PROGRAM Systemzeit
VAR
	fbFB_LocalSystemTime: FB_LocalSystemTime;
	fbGETSYSTEMTIME		: GETSYSTEMTIME;
    sNetID     			: T_AmsNetID := '';
    bEnable    			: BOOL := 1;
    dwCycle    			: DWORD(1..86400) := 5;
    dwOpt      			: DWORD := 1;
    tTimeout   			: TIME := DEFAULT_ADS_TIMEOUT;
	//bValid     		: BOOL := FALSE; GVL
	//dtsystemTime		: DATE_AND_TIME; GVL
	tzID       			: E_TimeZoneID := eTimeZoneID_Invalid;
END_VAR
VAR_INPUT
    systemTime 			: TIMESTRUCT;
END_VAR
VAR_OUTPUT
	
END_VAR

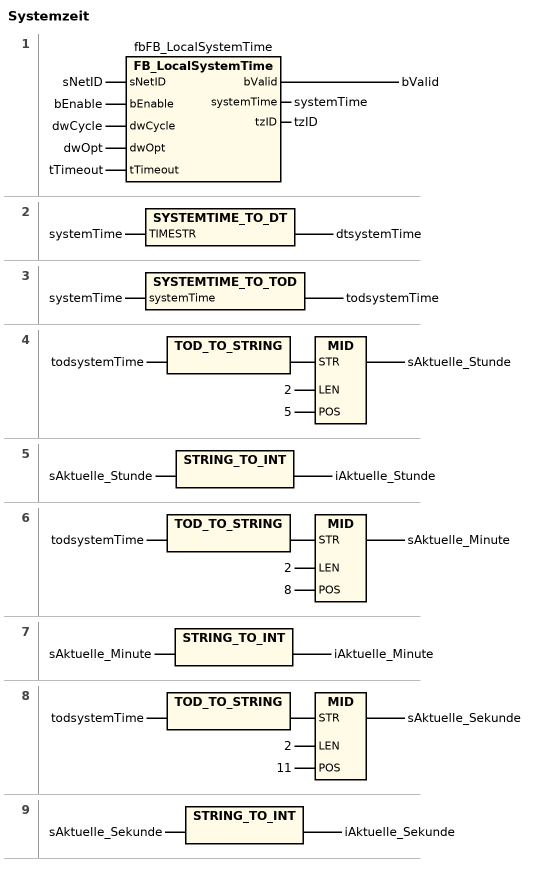
// NETWORK 1
fbFB_LocalSystemTime(
    sNetID := sNetID,
    bEnable := bEnable,
    dwCycle := dwCycle,
    dwOpt := dwOpt,
    tTimeout := tTimeout,
    systemTime => systemTime,
    tzID => tzID); // FB_LocalSystemTime
bValid := fbFB_LocalSystemTime.bValid;

// NETWORK 2
dtsystemTime := SYSTEMTIME_TO_DT(TIMESTR := systemTime);

// NETWORK 3
todsystemTime := SYSTEMTIME_TO_TOD(systemTime := systemTime);

// NETWORK 4
sAktuelle_Stunde := MID(STR := TOD_TO_STRING(todsystemTime), LEN := 2, POS := 5);

// NETWORK 5
iAktuelle_Stunde := STRING_TO_INT(sAktuelle_Stunde);

// NETWORK 6
sAktuelle_Minute := MID(STR := TOD_TO_STRING(todsystemTime), LEN := 2, POS := 8);

// NETWORK 7
iAktuelle_Minute := STRING_TO_INT(sAktuelle_Minute);

// NETWORK 8
sAktuelle_Sekunde := MID(STR := TOD_TO_STRING(todsystemTime), LEN := 2, POS := 11);

// NETWORK 9
iAktuelle_Sekunde := STRING_TO_INT(sAktuelle_Sekunde);

END_PROGRAM

(* stored: Version 1.1.0.1
   POU Systemzeit: Id {16b100f0-5455-4be7-a30b-12fa861a26a3}, SpecialFunc None *)
